// TIA Portal V21 export
FUNCTION "SimulaDoppioCilindroLineare" : Void   // FC29, LAD
{ S7_Optimized_Access := 'TRUE' }
// stored: SetENOAutomatically false
   VAR_INPUT
      CorsaCilindroAnteriore : Real;   // mm / %
      CorsaCilindroPosteriore : Real;   // mm / %
      K_Valvola_Anterirore : Int;   // K_Valvola che simula posizione anteriore
      K_Valvola_Posteriore : Int;   // K_Valvola che simula posizione posteriore
      K_Valvola_DoppioEffetto : Int;   // K_Valvola che comanda la valvola fisica
   END_VAR
   VAR_TEMP
      QuotaRichiesta : Real;
      PosizioneAttuale : Real;
      NumeroValvoleInPos : Byte;
   END_VAR
BEGIN

REGION Network 1 (SCL)
   "Valvola".V[#K_Valvola_DoppioEffetto].Prm.TogliComandoDopoPos := True;


   #QuotaRichiesta := 0;
   #PosizioneAttuale := "Valvola".V[#K_Valvola_DoppioEffetto].In.Feedback_PosizioneAttuale;
   #NumeroValvoleInPos := 0;

   REGION Calcolo quota di posizionamento
       IF "Valvola".V[#K_Valvola_Anterirore].Out.CmdPos THEN
           #QuotaRichiesta += #CorsaCilindroAnteriore;
           #NumeroValvoleInPos += 1;
       END_IF;
       IF "Valvola".V[#K_Valvola_Posteriore].Out.CmdPos THEN
           #QuotaRichiesta += #CorsaCilindroPosteriore;
           #NumeroValvoleInPos += 1;
       END_IF;

       "PosSenzaDeadBand_DB"(PosRichiesta := #QuotaRichiesta,
                             PosAttuale := #PosizioneAttuale,
                             ForzaPos := #NumeroValvoleInPos = 2,
                             ForzaNeg := #NumeroValvoleInPos = 0,
                             Pos => "Valvola".V[#K_Valvola_DoppioEffetto].In.RichiestaAutoPos,
                             Neg => "Valvola".V[#K_Valvola_DoppioEffetto].In.RichiestaAutoNeg);
   END_REGION
END_REGION
END_FUNCTION
